// TIA Portal V19 export
VAR_GLOBAL   // PLC tag table "U2Em6_Input"
   trayAutomaticFeedingDetectionU2Em6 AT %I46.0 : Bool;   // Em110_ Plastic tray drum feed detection / Em110_塑胶托盘滚筒进料检测
END_VAR
